{attribute 'GeneratedUsingTerminal: EK1100-0000-0018'}
{attribute addProperty BoxType "EK1100-0000-0018"}
{attribute addProperty Id "Beckhoff_EL5xxxEK1122Beckhoff_EL5xxxEK1122_8332829C2A_0001_EL5001_0000_0000EL5001_0636DF9417A_0002_EL5001_0000_0001EL5001_0636DF9417A_0003_EL5001_0000_1016EL5001_E64801B617A_0004_EL5001_0000_1017EL5001_09076D6E22A_0005_EL5001_0000_1018EL5001_09076D6E22A_0006_EL5001_0000_1019EL5001_09076D6E22A_0007_EL5001_0000_1020EL5001_09076D6E22A_0008_EL5001_0000_1021EL5001_09076D6E22A_0009_EL5001_0010_0000EL5001_0636DF9417A_0010_EL5001_0011_0016EL5001_E4817D5030A_0011_EL5001_0011_0017EL5001_E4817D5030A_0012_EL5001_0011_0018EL5001_E4817D5030A_0013_EL5001_0011_0019EL5001_EE91931B29A_0014_EL5001_0011_0020EL5001_EE91931B29A_0015_EL5001_0090_0016EL5001_09076D6E22A_0016_EL5002_0000_0016EL5002_814B807B32A_0017_EL5002_0000_0017EL5002_814B807B32A_0018_EL5002_0000_0018EL5002_814B807B32A_0019_EL5002_0000_0019EL5002_814B807B32A_0020_EL5002_0000_0020EL5002_DD23D25934A_0021_EL5021_0000_0016EL5021_48AC66F834A_0022_EL5021_0000_0017EL5021_48AC66F834A_0023_EL5021_0000_0018EL5021_48AC66F834A_0024_EL5021_0000_0019EL5021_48AC66F834A_0025_EL5021_0000_0020EL5021_48AC66F834A_0026_EL5021_0000_0021EL5021_48AC66F834A_0027_EL5021_0000_0022EL5021_48AC66F834A_0028_EL5021_0090_0018EL5021_48AC66F834A_0029_EL5021_0090_0019EL5021_48AC66F834A_0030_EL5032_0000_0021EL5032_78E1629D40A_0031_EL5032_0000_0023EL5032_78E1629D40A_0032_EL5032_0000_0024EL5032_78E1629D40A_0033_EL5032_0000_0025EL5032_78E1629D40A_0034_EL5032_0000_0026EL5032_78E1629D40A_0035_EL5032_0000_0027EL5032_78E1629D40A_0036_EL5032_0090_0016EL5032_78E1629D40A_0037_EL5042_0000_0016EL5042_78E1629D40A_0038_EL5072_0000_0016EL5072_7E09DEEC62A_0039_EL5101_0000_0000EL5101_1834142F20A_0040_EL5101_0000_0001EL5101_2E6F274D20A_0041_EL5101_0000_1017EL5101_2E6F274D20A_0042_EL5101_0000_1018EL5101_2E6F274D20A_0043_EL5101_0000_1019EL5101_075142ED38A_0044_EL5101_0000_1020EL5101_FD2A0DB838A_0045_EL5101_0000_1021EL5101_FD2A0DB838A_0046_EL5101_0000_1022EL5101_FD2A0DB838A_0047_EL5101_0000_1023EL5101_EE4069E438A_0048_EL5101_0000_1024EL5101_EE4069E438A_0049_EL5101_0010_0016EL5101_A21C120335A_0050_EL5101_0010_0017EL5101_A21C120335A_0051_EL5101_0010_0018EL5101_A21C120335A_0052_EL5101_0010_0019EL5101_A21C120335A_0053_EL5101_0011_0016EL5101_30AA1CB545A_0054_EL5101_0090_0016EL5101_EE4069E438A_0055_EL5101_0090_0017EL5101_EE4069E438A_0056_EL5101_1006_1019EL5101_075142ED38A_0057_EL5101_1006_1020EL5101_FD2A0DB838A_0058_EL5101_1006_1021EL5101_FD2A0DB838A_0059_EL5101_1006_1022EL5101_FD2A0DB838A_0060_EL5101_1006_1023EL5101_FD2A0DB838A_0061_EL5151_0000_0016EL5151_323C40EB40A_0062_EL5102_0000_0016EL5102_266AD387104A_0063_EL5112_0000_0016EL5112_844156A158A_0064_EL5122_0000_0016EL5122_26DE273B72A_0065_EL5151_0000_0017EL5151_25F4BC9F42A_0066_EL5151_0000_0018EL5151_25F4BC9F42A_0067_EL5151_0000_0019EL5151_25F4BC9F42A_0068_EL5151_0000_0020EL5151_269DA56F36A_0069_EL5151_0000_0021EL5151_9EA4F13436A_0070_EL5151_0000_0022EL5151_9EA4F13436A_0071_EL5151_0000_0023EL5151_9EA4F13436A_0072_EL5151_0000_0024EL5151_9EA4F13436A_0073_EL5151_0000_0025EL5151_269DA56F36A_0074_EL5151_0000_0026EL5151_269DA56F36A_0075_EL5151_0021_0018EL5151_0E726DD159A_0076_EL5151_0080_0016EL5151_FBCF8D4B36A_0077_EL5151_0080_0017EL5151_269DA56F36A_0078_EL5151_0080_0018EL5151_269DA56F36A_0079_EL5151_0080_0019EL5151_269DA56F36A_0080_EL5151_0080_0020EL5151_269DA56F36A_0081_EL5151_0080_0021EL5151_269DA56F36A_0082_EL5151_0090_0016EL5151_1214477B32A_0083_EL5152_0000_0016EL5152_ADEC432F42A_0084_EL5152_0000_0017EL5152_ADEC432F42A_0085_EL5152_0000_0018EL5152_B61CAFEE42A_0086_EL5152_0000_0019EL5152_B61CAFEE42"}
{attribute addProperty CRC "1370450550"}
{attribute addProperty Size "3086"}
TYPE Beckhoff_EL5xxx_51AF6A76 EXTENDS EK1100_AB5A9467 :
STRUCT
	{attribute addProperty Name "Beckhoff_EL5xxxEK1122"}
	{attribute addProperty PreviousPort "Beckhoff EL5xxx : B"}
	Beckhoff_EL5xxxEK1122 : Beckhoff_EL5xxxEK1122_8332829C;
	{attribute addProperty Name "A_0001_EL5001_0000_0000"}
	{attribute addProperty PreviousPort "Beckhoff EL5xxxEK1122 : C"}
	A_0001_EL5001_0000_0000 : EL5001_0636DF94;
	{attribute addProperty Name "A_0002_EL5001_0000_0001"}
	{attribute addProperty PreviousPort "A_0001(EL5001-0000-0000) : B"}
	A_0002_EL5001_0000_0001 : EL5001_0636DF94;
	{attribute addProperty Name "A_0003_EL5001_0000_1016"}
	{attribute addProperty PreviousPort "A_0002(EL5001-0000-0001) : B"}
	A_0003_EL5001_0000_1016 : EL5001_E64801B6;
	{attribute addProperty Name "A_0004_EL5001_0000_1017"}
	{attribute addProperty PreviousPort "A_0003(EL5001-0000-1016) : B"}
	A_0004_EL5001_0000_1017 : EL5001_09076D6E;
	{attribute addProperty Name "A_0005_EL5001_0000_1018"}
	{attribute addProperty PreviousPort "A_0004(EL5001-0000-1017) : B"}
	A_0005_EL5001_0000_1018 : EL5001_09076D6E;
	{attribute addProperty Name "A_0006_EL5001_0000_1019"}
	{attribute addProperty PreviousPort "A_0005(EL5001-0000-1018) : B"}
	A_0006_EL5001_0000_1019 : EL5001_09076D6E;
	{attribute addProperty Name "A_0007_EL5001_0000_1020"}
	{attribute addProperty PreviousPort "A_0006(EL5001-0000-1019) : B"}
	A_0007_EL5001_0000_1020 : EL5001_09076D6E;
	{attribute addProperty Name "A_0008_EL5001_0000_1021"}
	{attribute addProperty PreviousPort "A_0007(EL5001-0000-1020) : B"}
	A_0008_EL5001_0000_1021 : EL5001_09076D6E;
	{attribute addProperty Name "A_0009_EL5001_0010_0000"}
	{attribute addProperty PreviousPort "A_0008(EL5001-0000-1021) : B"}
	A_0009_EL5001_0010_0000 : EL5001_0636DF94;
	{attribute addProperty Name "A_0010_EL5001_0011_0016"}
	{attribute addProperty PreviousPort "A_0009(EL5001-0010-0000) : B"}
	A_0010_EL5001_0011_0016 : EL5001_E4817D50;
	{attribute addProperty Name "A_0011_EL5001_0011_0017"}
	{attribute addProperty PreviousPort "A_0010(EL5001-0011-0016) : B"}
	A_0011_EL5001_0011_0017 : EL5001_E4817D50;
	{attribute addProperty Name "A_0012_EL5001_0011_0018"}
	{attribute addProperty PreviousPort "A_0011(EL5001-0011-0017) : B"}
	A_0012_EL5001_0011_0018 : EL5001_E4817D50;
	{attribute addProperty Name "A_0013_EL5001_0011_0019"}
	{attribute addProperty PreviousPort "A_0012(EL5001-0011-0018) : B"}
	A_0013_EL5001_0011_0019 : EL5001_EE91931B;
	{attribute addProperty Name "A_0014_EL5001_0011_0020"}
	{attribute addProperty PreviousPort "A_0013(EL5001-0011-0019) : B"}
	A_0014_EL5001_0011_0020 : EL5001_EE91931B;
	{attribute addProperty Name "A_0015_EL5001_0090_0016"}
	{attribute addProperty PreviousPort "A_0014(EL5001-0011-0020) : B"}
	A_0015_EL5001_0090_0016 : EL5001_09076D6E;
	{attribute addProperty Name "A_0016_EL5002_0000_0016"}
	{attribute addProperty PreviousPort "A_0015(EL5001-0090-0016) : B"}
	A_0016_EL5002_0000_0016 : EL5002_814B807B;
	{attribute addProperty Name "A_0017_EL5002_0000_0017"}
	{attribute addProperty PreviousPort "A_0016(EL5002-0000-0016) : B"}
	A_0017_EL5002_0000_0017 : EL5002_814B807B;
	{attribute addProperty Name "A_0018_EL5002_0000_0018"}
	{attribute addProperty PreviousPort "A_0017(EL5002-0000-0017) : B"}
	A_0018_EL5002_0000_0018 : EL5002_814B807B;
	{attribute addProperty Name "A_0019_EL5002_0000_0019"}
	{attribute addProperty PreviousPort "A_0018(EL5002-0000-0018) : B"}
	A_0019_EL5002_0000_0019 : EL5002_814B807B;
	{attribute addProperty Name "A_0020_EL5002_0000_0020"}
	{attribute addProperty PreviousPort "A_0019(EL5002-0000-0019) : B"}
	A_0020_EL5002_0000_0020 : EL5002_DD23D259;
	{attribute addProperty Name "A_0021_EL5021_0000_0016"}
	{attribute addProperty PreviousPort "A_0020(EL5002-0000-0020) : B"}
	A_0021_EL5021_0000_0016 : EL5021_48AC66F8;
	{attribute addProperty Name "A_0022_EL5021_0000_0017"}
	{attribute addProperty PreviousPort "A_0021(EL5021-0000-0016) : B"}
	A_0022_EL5021_0000_0017 : EL5021_48AC66F8;
	{attribute addProperty Name "A_0023_EL5021_0000_0018"}
	{attribute addProperty PreviousPort "A_0022(EL5021-0000-0017) : B"}
	A_0023_EL5021_0000_0018 : EL5021_48AC66F8;
	{attribute addProperty Name "A_0024_EL5021_0000_0019"}
	{attribute addProperty PreviousPort "A_0023(EL5021-0000-0018) : B"}
	A_0024_EL5021_0000_0019 : EL5021_48AC66F8;
	{attribute addProperty Name "A_0025_EL5021_0000_0020"}
	{attribute addProperty PreviousPort "A_0024(EL5021-0000-0019) : B"}
	A_0025_EL5021_0000_0020 : EL5021_48AC66F8;
	{attribute addProperty Name "A_0026_EL5021_0000_0021"}
	{attribute addProperty PreviousPort "A_0025(EL5021-0000-0020) : B"}
	A_0026_EL5021_0000_0021 : EL5021_48AC66F8;
	{attribute addProperty Name "A_0027_EL5021_0000_0022"}
	{attribute addProperty PreviousPort "A_0026(EL5021-0000-0021) : B"}
	A_0027_EL5021_0000_0022 : EL5021_48AC66F8;
	{attribute addProperty Name "A_0028_EL5021_0090_0018"}
	{attribute addProperty PreviousPort "A_0027(EL5021-0000-0022) : B"}
	A_0028_EL5021_0090_0018 : EL5021_48AC66F8;
	{attribute addProperty Name "A_0029_EL5021_0090_0019"}
	{attribute addProperty PreviousPort "A_0028(EL5021-0090-0018) : B"}
	A_0029_EL5021_0090_0019 : EL5021_48AC66F8;
	{attribute addProperty Name "A_0030_EL5032_0000_0021"}
	{attribute addProperty PreviousPort "A_0029(EL5021-0090-0019) : B"}
	A_0030_EL5032_0000_0021 : EL5032_78E1629D;
	{attribute addProperty Name "A_0031_EL5032_0000_0023"}
	{attribute addProperty PreviousPort "A_0030(EL5032-0000-0021) : B"}
	A_0031_EL5032_0000_0023 : EL5032_78E1629D;
	{attribute addProperty Name "A_0032_EL5032_0000_0024"}
	{attribute addProperty PreviousPort "A_0031(EL5032-0000-0023) : B"}
	A_0032_EL5032_0000_0024 : EL5032_78E1629D;
	{attribute addProperty Name "A_0033_EL5032_0000_0025"}
	{attribute addProperty PreviousPort "A_0032(EL5032-0000-0024) : B"}
	A_0033_EL5032_0000_0025 : EL5032_78E1629D;
	{attribute addProperty Name "A_0034_EL5032_0000_0026"}
	{attribute addProperty PreviousPort "A_0033(EL5032-0000-0025) : B"}
	A_0034_EL5032_0000_0026 : EL5032_78E1629D;
	{attribute addProperty Name "A_0035_EL5032_0000_0027"}
	{attribute addProperty PreviousPort "A_0034(EL5032-0000-0026) : B"}
	A_0035_EL5032_0000_0027 : EL5032_78E1629D;
	{attribute addProperty Name "A_0036_EL5032_0090_0016"}
	{attribute addProperty PreviousPort "A_0035(EL5032-0000-0027) : B"}
	A_0036_EL5032_0090_0016 : EL5032_78E1629D;
	{attribute addProperty Name "A_0037_EL5042_0000_0016"}
	{attribute addProperty PreviousPort "A_0036(EL5032-0090-0016) : B"}
	A_0037_EL5042_0000_0016 : EL5042_78E1629D;
	{attribute addProperty Name "A_0038_EL5072_0000_0016"}
	{attribute addProperty PreviousPort "A_0037(EL5042-0000-0016) : B"}
	A_0038_EL5072_0000_0016 : EL5072_7E09DEEC;
	{attribute addProperty Name "A_0039_EL5101_0000_0000"}
	{attribute addProperty PreviousPort "A_0038(EL5072-0000-0016) : B"}
	A_0039_EL5101_0000_0000 : EL5101_1834142F;
	{attribute addProperty Name "A_0040_EL5101_0000_0001"}
	{attribute addProperty PreviousPort "A_0039(EL5101-0000-0000) : B"}
	A_0040_EL5101_0000_0001 : EL5101_2E6F274D;
	{attribute addProperty Name "A_0041_EL5101_0000_1017"}
	{attribute addProperty PreviousPort "A_0040(EL5101-0000-0001) : B"}
	A_0041_EL5101_0000_1017 : EL5101_2E6F274D;
	{attribute addProperty Name "A_0042_EL5101_0000_1018"}
	{attribute addProperty PreviousPort "A_0041(EL5101-0000-1017) : B"}
	A_0042_EL5101_0000_1018 : EL5101_2E6F274D;
	{attribute addProperty Name "A_0043_EL5101_0000_1019"}
	{attribute addProperty PreviousPort "A_0042(EL5101-0000-1018) : B"}
	A_0043_EL5101_0000_1019 : EL5101_075142ED;
	{attribute addProperty Name "A_0044_EL5101_0000_1020"}
	{attribute addProperty PreviousPort "A_0043(EL5101-0000-1019) : B"}
	A_0044_EL5101_0000_1020 : EL5101_FD2A0DB8;
	{attribute addProperty Name "A_0045_EL5101_0000_1021"}
	{attribute addProperty PreviousPort "A_0044(EL5101-0000-1020) : B"}
	A_0045_EL5101_0000_1021 : EL5101_FD2A0DB8;
	{attribute addProperty Name "A_0046_EL5101_0000_1022"}
	{attribute addProperty PreviousPort "A_0045(EL5101-0000-1021) : B"}
	A_0046_EL5101_0000_1022 : EL5101_FD2A0DB8;
	{attribute addProperty Name "A_0047_EL5101_0000_1023"}
	{attribute addProperty PreviousPort "A_0046(EL5101-0000-1022) : B"}
	A_0047_EL5101_0000_1023 : EL5101_EE4069E4;
	{attribute addProperty Name "A_0048_EL5101_0000_1024"}
	{attribute addProperty PreviousPort "A_0047(EL5101-0000-1023) : B"}
	A_0048_EL5101_0000_1024 : EL5101_EE4069E4;
	{attribute addProperty Name "A_0049_EL5101_0010_0016"}
	{attribute addProperty PreviousPort "A_0048(EL5101-0000-1024) : B"}
	A_0049_EL5101_0010_0016 : EL5101_A21C1203;
	{attribute addProperty Name "A_0050_EL5101_0010_0017"}
	{attribute addProperty PreviousPort "A_0049(EL5101-0010-0016) : B"}
	A_0050_EL5101_0010_0017 : EL5101_A21C1203;
	{attribute addProperty Name "A_0051_EL5101_0010_0018"}
	{attribute addProperty PreviousPort "A_0050(EL5101-0010-0017) : B"}
	A_0051_EL5101_0010_0018 : EL5101_A21C1203;
	{attribute addProperty Name "A_0052_EL5101_0010_0019"}
	{attribute addProperty PreviousPort "A_0051(EL5101-0010-0018) : B"}
	A_0052_EL5101_0010_0019 : EL5101_A21C1203;
	{attribute addProperty Name "A_0053_EL5101_0011_0016"}
	{attribute addProperty PreviousPort "A_0052(EL5101-0010-0019) : B"}
	A_0053_EL5101_0011_0016 : EL5101_30AA1CB5;
	{attribute addProperty Name "A_0054_EL5101_0090_0016"}
	{attribute addProperty PreviousPort "A_0053(EL5101-0011-0016) : B"}
	A_0054_EL5101_0090_0016 : EL5101_EE4069E4;
	{attribute addProperty Name "A_0055_EL5101_0090_0017"}
	{attribute addProperty PreviousPort "A_0054(EL5101-0090-0016) : B"}
	A_0055_EL5101_0090_0017 : EL5101_EE4069E4;
	{attribute addProperty Name "A_0056_EL5101_1006_1019"}
	{attribute addProperty PreviousPort "A_0055(EL5101-0090-0017) : B"}
	A_0056_EL5101_1006_1019 : EL5101_075142ED;
	{attribute addProperty Name "A_0057_EL5101_1006_1020"}
	{attribute addProperty PreviousPort "A_0056(EL5101-1006-1019) : B"}
	A_0057_EL5101_1006_1020 : EL5101_FD2A0DB8;
	{attribute addProperty Name "A_0058_EL5101_1006_1021"}
	{attribute addProperty PreviousPort "A_0057(EL5101-1006-1020) : B"}
	A_0058_EL5101_1006_1021 : EL5101_FD2A0DB8;
	{attribute addProperty Name "A_0059_EL5101_1006_1022"}
	{attribute addProperty PreviousPort "A_0058(EL5101-1006-1021) : B"}
	A_0059_EL5101_1006_1022 : EL5101_FD2A0DB8;
	{attribute addProperty Name "A_0060_EL5101_1006_1023"}
	{attribute addProperty PreviousPort "A_0059(EL5101-1006-1022) : B"}
	A_0060_EL5101_1006_1023 : EL5101_FD2A0DB8;
	{attribute addProperty Name "A_0061_EL5151_0000_0016"}
	{attribute addProperty PreviousPort "A_0060(EL5101-1006-1023) : B"}
	A_0061_EL5151_0000_0016 : EL5151_323C40EB;
	{attribute addProperty Name "A_0062_EL5102_0000_0016"}
	{attribute addProperty PreviousPort "A_0061(EL5151-0000-0016) : B"}
	A_0062_EL5102_0000_0016 : EL5102_266AD387;
	{attribute addProperty Name "A_0063_EL5112_0000_0016"}
	{attribute addProperty PreviousPort "A_0062(EL5102-0000-0016) : B"}
	A_0063_EL5112_0000_0016 : EL5112_844156A1;
	{attribute addProperty Name "A_0064_EL5122_0000_0016"}
	{attribute addProperty PreviousPort "A_0063(EL5112-0000-0016) : B"}
	A_0064_EL5122_0000_0016 : EL5122_26DE273B;
	{attribute addProperty Name "A_0065_EL5151_0000_0017"}
	{attribute addProperty PreviousPort "A_0064(EL5122-0000-0016) : B"}
	A_0065_EL5151_0000_0017 : EL5151_25F4BC9F;
	{attribute addProperty Name "A_0066_EL5151_0000_0018"}
	{attribute addProperty PreviousPort "A_0065(EL5151-0000-0017) : B"}
	A_0066_EL5151_0000_0018 : EL5151_25F4BC9F;
	{attribute addProperty Name "A_0067_EL5151_0000_0019"}
	{attribute addProperty PreviousPort "A_0066(EL5151-0000-0018) : B"}
	A_0067_EL5151_0000_0019 : EL5151_25F4BC9F;
	{attribute addProperty Name "A_0068_EL5151_0000_0020"}
	{attribute addProperty PreviousPort "A_0067(EL5151-0000-0019) : B"}
	A_0068_EL5151_0000_0020 : EL5151_269DA56F;
	{attribute addProperty Name "A_0069_EL5151_0000_0021"}
	{attribute addProperty PreviousPort "A_0068(EL5151-0000-0020) : B"}
	A_0069_EL5151_0000_0021 : EL5151_9EA4F134;
	{attribute addProperty Name "A_0070_EL5151_0000_0022"}
	{attribute addProperty PreviousPort "A_0069(EL5151-0000-0021) : B"}
	A_0070_EL5151_0000_0022 : EL5151_9EA4F134;
	{attribute addProperty Name "A_0071_EL5151_0000_0023"}
	{attribute addProperty PreviousPort "A_0070(EL5151-0000-0022) : B"}
	A_0071_EL5151_0000_0023 : EL5151_9EA4F134;
	{attribute addProperty Name "A_0072_EL5151_0000_0024"}
	{attribute addProperty PreviousPort "A_0071(EL5151-0000-0023) : B"}
	A_0072_EL5151_0000_0024 : EL5151_9EA4F134;
	{attribute addProperty Name "A_0073_EL5151_0000_0025"}
	{attribute addProperty PreviousPort "A_0072(EL5151-0000-0024) : B"}
	A_0073_EL5151_0000_0025 : EL5151_269DA56F;
	{attribute addProperty Name "A_0074_EL5151_0000_0026"}
	{attribute addProperty PreviousPort "A_0073(EL5151-0000-0025) : B"}
	A_0074_EL5151_0000_0026 : EL5151_269DA56F;
	{attribute addProperty Name "A_0075_EL5151_0021_0018"}
	{attribute addProperty PreviousPort "A_0074(EL5151-0000-0026) : B"}
	A_0075_EL5151_0021_0018 : EL5151_0E726DD1;
	{attribute addProperty Name "A_0076_EL5151_0080_0016"}
	{attribute addProperty PreviousPort "A_0075(EL5151-0021-0018) : B"}
	A_0076_EL5151_0080_0016 : EL5151_FBCF8D4B;
	{attribute addProperty Name "A_0077_EL5151_0080_0017"}
	{attribute addProperty PreviousPort "A_0076(EL5151-0080-0016) : B"}
	A_0077_EL5151_0080_0017 : EL5151_269DA56F;
	{attribute addProperty Name "A_0078_EL5151_0080_0018"}
	{attribute addProperty PreviousPort "A_0077(EL5151-0080-0017) : B"}
	A_0078_EL5151_0080_0018 : EL5151_269DA56F;
	{attribute addProperty Name "A_0079_EL5151_0080_0019"}
	{attribute addProperty PreviousPort "A_0078(EL5151-0080-0018) : B"}
	A_0079_EL5151_0080_0019 : EL5151_269DA56F;
	{attribute addProperty Name "A_0080_EL5151_0080_0020"}
	{attribute addProperty PreviousPort "A_0079(EL5151-0080-0019) : B"}
	A_0080_EL5151_0080_0020 : EL5151_269DA56F;
	{attribute addProperty Name "A_0081_EL5151_0080_0021"}
	{attribute addProperty PreviousPort "A_0080(EL5151-0080-0020) : B"}
	A_0081_EL5151_0080_0021 : EL5151_269DA56F;
	{attribute addProperty Name "A_0082_EL5151_0090_0016"}
	{attribute addProperty PreviousPort "A_0081(EL5151-0080-0021) : B"}
	A_0082_EL5151_0090_0016 : EL5151_1214477B;
	{attribute addProperty Name "A_0083_EL5152_0000_0016"}
	{attribute addProperty PreviousPort "A_0082(EL5151-0090-0016) : B"}
	A_0083_EL5152_0000_0016 : EL5152_ADEC432F;
	{attribute addProperty Name "A_0084_EL5152_0000_0017"}
	{attribute addProperty PreviousPort "A_0083(EL5152-0000-0016) : B"}
	A_0084_EL5152_0000_0017 : EL5152_ADEC432F;
	{attribute addProperty Name "A_0085_EL5152_0000_0018"}
	{attribute addProperty PreviousPort "A_0084(EL5152-0000-0017) : B"}
	A_0085_EL5152_0000_0018 : EL5152_B61CAFEE;
	{attribute addProperty Name "A_0086_EL5152_0000_0019"}
	{attribute addProperty PreviousPort "A_0085(EL5152-0000-0018) : B"}
	A_0086_EL5152_0000_0019 : EL5152_B61CAFEE;
END_STRUCT
END_TYPE

(* stored: Version 1.2.0.0, ProductVersion 3.1.4024.9
   DUT Beckhoff_EL5xxx_51AF6A76: Id {84a2f249-437e-433f-bfc8-5f59e5c2fdcb} *)
